// TIA Portal V17 export
// export: Created 2024-09-02T12:50:26.4768897Z, ExportSetting WithDefaults, DisplayName Totally Integrated Automation Portal, DisplayVersion V17, DisplayName TIA Portal Openness, DisplayVersion V17, DisplayName TIA Portal Version Control Interface, DisplayVersion V17, DisplayName STEP 7 Professional, DisplayVersion V17, DisplayName STEP 7 Safety, DisplayVersion V17, DisplayName WinCC Professional, DisplayVersion V17
TYPE "TypeSationsSum"
// stored: IsFailsafeCompliant false
   STRUCT
      Transport_Running : Bool;   // Anzeige Transport läuft / Display Transport running
      Screen_No_active : Int;   // 296
      ExternalDevice : Array[1..10] of Struct   // Fremdgeräte / Foreign devices
         State : Int;
      END_STRUCT;
      Station : Array[1..4] of Struct   // Station uebersicht / Station overview
         Status : Struct
            Display : Bool;
            EStop : Bool;
            Fault : Bool;
            SafetyDoor : Bool;
            SpecialFunction : Bool;
            Home : Bool;
            Done { ExternalWritable := 'False'} : Bool;
         END_STRUCT;
      END_STRUCT;
      SLG_Display : Array[1..8] of Struct   // SLG Anzeige / SLG Display
         State : Int;   // 1=einblenden;2=gelesen;3=geschrieben;4=Störung / 1 = insert, 2 = Read, 3 = written, 4 = OK, 5 = Error
      END_STRUCT;
      HardwareDiagnose : Struct   // Zustandsanzeige Hardwarediagnose / Status display Hardware diagnostics
         StatusDisplay_Safety : Byte;   // Zustandsanzeige Safety / Status display Safety
         StatusDisplay_Reserve : Byte;   // Zustandsanzeige Reserve / Status display Reserve
         StatusDisplay_PB_PN : Byte;   // Zustandsanzeige Profibus / Profinet / Status display Profibus / Profinet
         StatusDisplay_611U : Byte;   // Zustandsanzeige 611U / Status display 611U
         StatusDisplay_Moby : Byte;   // Zustandsanzeige Moby / Status display Moby
         StatusDisplay_ASI : Byte;   // Zustandsanzeige AS Interface / Status display AS Interface
      END_STRUCT;
      PartCounter : Struct   // Stuckzahl / Quantity
         Layer_1_HM : Bool;
         Layer_1_fp : Bool;
         Layer_2_HM : Bool;
         Layer_2_fp : Bool;
         Layer_3_HM : Bool;
         Layer_3_fp : Bool;
         Tag_HM : Bool;
         Tag_fp : Bool;
         Tag_old : Byte;
         "Type" : Byte;
      END_STRUCT;
      Function : Struct   // Sonderfunktionen / Special features
         SafetyDoor : Struct   // Anforderung Schutztueren / Requirement of Safety Door
            ButtonDisplay : Int;   // Button Anzeige Gestaltung / Button Display Design
            active : Bool;   // Button aktiv (gedrückt) / Button active (pressed)
         END_STRUCT;
         TypeAck : Struct   // Anforderung Typ quittieren / Requirement of Typ acknowledgement
            ButtonDisplay : Int;   // Button Anzeige Gestaltung / Button Display Design
            active : Bool;   // Button aktiv (gedrückt) / Button active (pressed)
         END_STRUCT;
         SafetyDoor_2 : Struct   // Anforderung Schutztueren / Requirement of Safety Door
            ButtonDisplay : Int;   // Button Anzeige Gestaltung / Button Display Design
            active : Bool;   // Button aktiv (gedrückt) / Button active (pressed)
         END_STRUCT;
         _4 : Struct   // Funktion Frei / Function Free
            ButtonDisplay : Int;   // Button Anzeige Gestaltung / Button Display Design
            active : Bool;   // Button aktiv (gedrückt) / Button active (pressed)
         END_STRUCT;
         _5 : Struct   // Funktion Frei / Function Free
            ButtonDisplay : Int;   // Button Anzeige Gestaltung / Button Display Design
            active : Bool;   // Button aktiv (gedrückt) / Button active (pressed)
         END_STRUCT;
         _6 : Struct   // Funktion Frei / Function Free
            ButtonDisplay : Int;   // Button Anzeige Gestaltung / Button Display Design
            active : Bool;   // Button aktiv (gedrückt) / Button active (pressed)
         END_STRUCT;
         _7 : Struct   // Funktion Frei / Function Free
            ButtonDisplay : Int;   // Button Anzeige Gestaltung / Button Display Design
            active : Bool;   // Button aktiv (gedrückt) / Button active (pressed)
         END_STRUCT;
         _8 : Struct   // Funktion Frei / Function Free
            ButtonDisplay : Int;   // Button Anzeige Gestaltung / Button Display Design
            active : Bool;   // Button aktiv (gedrückt) / Button active (pressed)
         END_STRUCT;
      END_STRUCT;
   END_STRUCT;
END_TYPE
